(* CODESYS project ctrlxVirtual.export

Project tree, tasks and I/O mapping:
  Device : ctrlX COREvirtual, Bosch Rexroth AG, order no. dependent on customer specific configuration, version 1.14.0.0
    application Application
      libraries: ; SampleSchema, 0.0.1 (Bosch Rexroth)
      task MainTask (cyclic, interval 200 ms, priority 30) calls PLC_PRG
      CheckFunctions/
        function CheckDivDInt [ST]
        function CheckDivLInt [ST]
        function CheckDivLReal [ST]
        function CheckDivReal [ST]
        function CheckLRangeSigned [ST]
        function CheckLRangeUnsigned [ST]
        function CheckRangeSigned [ST]
        function CheckRangeUnsigned [ST]
        function CheckBounds [ST]
        function CheckPointer [ST]
      program PLC_PRG [ST]
    Realtime_Data : DataLayer, Bosch Rexroth AG, version 1.8.0.0
*)

// Device/Application/PLC_PRG
PROGRAM PLC_PRG
VAR
	bStart_read: BOOL := TRUE;
	bStart_write: BOOL;

	// Read values
	bExecute_read: BOOL;
	fbDL_ReadNodeValue: sampleSchema.DL_ReadNodeValue;
	bActive_read: BOOL;
	bDone_read: BOOL;
	
	DataRead: sampleSchema.DL_NodeValue;
	bErrorRead: BOOL;
	ErrorIDRead: ERROR_CODE;
	ErrorIdent_read: ERROR_STRUCT;

	fbR_TRIG_read: R_TRIG;

	fbFlatbuffer : sampleSchema.sample_schema_InertialValue;

	iRead_X: INT;
	iRead_Y: INT;
	iRead_Z: INT;
	iRead: INT;
	
	///Write values
	fbBuilder: sampleSchema.FlatBufferBuilder();
	
	iWrite_X: INT;
	iWrite_Y: INT;
	iWrite_Z: INT;
	iWritten: INT;
	
	bExecute_write: BOOL;
	fbDL_WriteNodeValue: sampleSchema.DL_WriteNodeValue;
	bActive_write: BOOL;
	bDone_write: BOOL;
	fbValueIn: sampleSchema.DL_NodeValue;
	fbValueOut: sampleSchema.DL_NodeValue;
	bError_write: BOOL;
	ErrorID_write: ERROR_CODE;
	ErrorIdent_write: ERROR_STRUCT;
	
	fbR_TRIG_write: R_TRIG;
	

	strNodePath: STRING(255) := 'sdk-cpp-alldata/dynamic/fbs';
	
END_VAR

IF bStart_read THEN
	bStart_read := FALSE;
	bExecute_read := TRUE;	
END_IF


fbDL_ReadNodeValue(
	Execute:= bExecute_read,
	Done=> bDone_read,
	Active=> bActive_read,
	Error=> bErrorRead,
	ErrorID=> ErrorIDRead,
	ErrorIdent=> ErrorIdent_read,
	ClientId:= ,
	NodeName:= strNodePath,
	NodeValue:= DataRead);

IF bDone_read AND bExecute_read THEN
	bExecute_read := FALSE;

	fbFlatbuffer.getRootAsInertialValue(data:=
	DataRead.GetData(), size:= DataRead.GetSize());
	
	iRead_X := fbFlatbuffer.getX();
	iRead_Y := fbFlatbuffer.getY();
	iRead_Z := fbFlatbuffer.getZ();	
	iRead := iRead + 1;
		
	bStart_write := TRUE;
END_IF

	
IF bStart_write THEN
	bStart_write := FALSE;

	iWrite_X := iRead_X + 100;
	iWrite_Y := iRead_Y + 100;
	iWrite_Z := iRead_Z + 100;

	fbBuilder(forceDefaults := TRUE);
	fbFlatbuffer.startInertialValue(fbBuilder);
	fbFlatbuffer.addX(iWrite_X);
	fbFlatbuffer.addY(iWrite_Y);
	fbFlatbuffer.addZ(iWrite_Z);
	fbBuilder.finish(fbFlatbuffer.endInertialValue());
	fbValueIn.SetFlatbuffer(fbBuilder);
	
	bExecute_write := TRUE;
END_IF

	
fbDL_WriteNodeValue(
	Execute:= bExecute_write,
	Done=> bDone_write,
	Active=> bActive_write,
	Error=> bError_write,
	ErrorID=> ErrorID_write,
	ErrorIdent=> ErrorIdent_write,
	ClientId:= ,
	NodeName:= strNodePath,
	NodeValueIn:= fbValueIn,
	NodeValueOut:= fbValueOut);

IF bDone_write AND bExecute_write THEN
	bExecute_write := FALSE;	
	iWritten := iWritten + 1;
	
	bStart_read := TRUE;
END_IF

END_PROGRAM

// Device/Application/CheckFunctions/CheckDivDInt
// Short description:        Test function to increase machine safety by detecting unauthorized division by zero of INT, UINT, DINT, UDINT, WORD and DWORD variables
// 
// Functional description:   This function will be called implicitly before the division takes places.
//                           The divisor will be checked for 0.
//                           In case of 0, an error is entered in the plc logger and the application is stopped due to an access violation to avoid machine damage.
//                           In this case, check the callstack (menu Debug/Callstack) and modify the faulty logic. 
// 
// Handling particularities: This function increases the cycle time of all tasks using divisions.
//                           The increase depends on the number of the divisions.
//                           After inserting/removing this function, no online-change will be possible! 
//                           A complete download will be necessary!
//                           The implementation has to be adjusted to your application/machine.
//                           In case of a division by zero, the PLC-Task will generate an access violation which leads to an application stop.
//                           Please verify whether this default behaviour can damage your machine or lead to a complex recommissioning. 
//                           In this case, adapt the error reaction to your application.
//                          
//                           If your application isn't too time-critical, you should leave this function whil comissioning the machine and production in your application.  
//                           If you remove this function, ensure that your code is faultless.
//                          
// Do not change the declaration of this function! Add only local variables.  
// Do not change the attributes above the function header!
{attribute 'check_div_int32'}
{attribute 'no_check'}
{attribute 'signature_flag' := '1073741824'}
FUNCTION CheckDivDInt : DINT
VAR_INPUT
  divisor: DINT; // Divisor of the division
END_VAR
VAR
  ptNull: POINTER TO BYTE := 0; // Nullpointer for triggering an access violation
  strError: STRING;             // Diagnostic text for the PLC logger entry
END_VAR

    (**************************************************************************************************)
    (* The implementation has to be adjusted to your application/machine.                             *)
    (* This is an exemplary implementation of the function.                                           *)
    (* Per default, an access violation is generated to avoid machine damage                          *)
    (* Check the Call Stack (menu Debug/Callstack) and modify the faulty logic!                       *)
    (**************************************************************************************************)

IF divisor = 0 THEN
  strError:= 'CheckDivDInt: Invalid division by 0 - check the callstack';
//  Default implementation for APPLICATION WILL BE STOPPED: 
//  Set an error into the plc logger
  LogAdd2(hLogger:= CmpLog.LOG_STD_LOGGER,udiCmpID:= 16#1000,udiClassID:= LogClass.LOG_ERROR,udiErrorID:= 1,udiInfoID:= 1,pszInfo:= strError);
//  Triggering an access violation --> Application will be stopped
  ptNull^ := 0;(* Triggering an access violation *)

// // Example for APPLICATION WILL NOT BE STOPPED:
// // Set the divisor to 1 
// //   --> no access violation (div by zero) will be triggered
// //   --> keep PLC-task running 
// // Set a warning into the plc logger
// // NOTE: There is still an implementation error in your application code!
// 
//  LogAdd2(hLogger:= CmpLog.LOG_STD_LOGGER,udiCmpID:= 16#1000,udiClassID:= LogClass.LOG_WARNING,udiErrorID:= 1,udiInfoID:= 1,pszInfo:= strError);
//  CheckDivDint := 1; //Division by 1 instead of zero 
//  return;	

ELSE // division is ok
  CheckDivDInt:=divisor;
END_IF;

END_FUNCTION

// Device/Application/CheckFunctions/CheckDivLInt
// Short description:        Test function to increase machine safety by detecting unauthorized division by zero of LINT, ULINT and LWORD variables
// 
// Functional description:   This function will be called implicitly before the division takes places.
//                           The divisor will be checked for 0.
//                           In case of 0, an error is entered in the plc logger and the application is stopped due to an access violation to avoid machine damage.
//                           In this case, check the callstack (menu Debug/Callstack) and modify the faulty logic. 
// 
// Handling particularities: This function increases the cycle time of all tasks using divisions.
//                           The increase depends on the number of the divisions.
//                           After inserting/removing this function, no online-change will be possible! 
//                           A complete download will be necessary!
//                           The implementation has to be adjusted to your application/machine.
//                           In case of a division by zero, the PLC-Task will generate an access violation which leads to an application stop.
//                           Please verify whether this default behaviour can damage your machine or lead to a complex recommissioning. 
//                           In this case, adapt the error reaction to your application.
//                          
//                           If your application isn't too time-critical, you should leave this function whil comissioning the machine and production in your application.  
//                           If you remove this function, ensure that your code is faultless.
//                          
// Do not change the declaration of this function! Add only local variables.  
// Do not change the attributes above the function header!
{attribute 'check_div_int64'}
{attribute 'no_check'}
{attribute 'signature_flag' := '1073741824'}
FUNCTION CheckDivLInt : LINT
VAR_INPUT
  divisor: LINT; // Divisor of the division
END_VAR
VAR
  ptNull: POINTER TO BYTE := 0; // Nullpointer for triggering an access violation
  strError: STRING;             // Diagnostic text for the PLC logger entry
END_VAR

    (**************************************************************************************************)
    (* The implementation has to be adjusted to your application/machine.                             *)
    (* This is an exemplary implementation of the function.                                           *)
    (* Per default, an access violation is generated to avoid machine damage                          *)
    (* Check the Call Stack (menu Debug/Callstack) and modify the faulty logic!                       *)
    (**************************************************************************************************)

IF divisor = 0 THEN
  strError:= 'CheckDivLInt: Invalid division by 0 - check the callstack';
//  Default implementation for APPLICATION WILL BE STOPPED: 
//  Set an error into the plc logger
  LogAdd2(hLogger:= CmpLog.LOG_STD_LOGGER,udiCmpID:= 16#1000,udiClassID:= LogClass.LOG_ERROR,udiErrorID:= 1,udiInfoID:= 1,pszInfo:= strError);
//  Triggering an access violation --> Application will be stopped
  ptNull^ := 0;(* Triggering an access violation *)

// // Example for APPLICATION WILL NOT BE STOPPED:
// // Set the divisor to 1 
// //   --> no access violation (div by zero) will be triggered
// //   --> keep PLC-task running 
// // Set a warning into the plc logger
// // NOTE: There is still an implementation error in your application code!
//  
//  LogAdd2(hLogger:= CmpLog.LOG_STD_LOGGER,udiCmpID:= 16#1000,udiClassID:= LogClass.LOG_WARNING,udiErrorID:= 1,udiInfoID:= 1,pszInfo:= strError);
//  CheckDivLInt := 1; //Division by 1 instead of zero 
//  return;	

ELSE // division is ok
  CheckDivLInt:=divisor;
END_IF;

END_FUNCTION

// Device/Application/CheckFunctions/CheckDivLReal
// Short description:        Test function to increase machine safety by detecting unauthorized division by zero of variables of type LREAL
// 
// Functional description:   This function will be called implicitly before the division takes places.
//                           The divisor will be checked for 0.0.
//                           In case of 0.0, an error is entered in the plc logger and the application is stopped due to an access violation to avoid machine damage.
//                           In this case, check the callstack (menu Debug/Callstack) and modify the faulty logic. 
// 
// Handling particularities: This function increases the cycle time of all tasks using divisions.
//                           The increase depends on the number of the divisions.
//                           After inserting/removing this function, no online-change will be possible! 
//                           A complete download will be necessary!
//                           The implementation has to be adjusted to your application/machine.
//                           In case of a division by zero, the PLC-Task will generate an access violation which leads to an application stop.
//                           Please verify whether this default behaviour can damage your machine or lead to a complex recommissioning. 
//                           In this case, adapt the error reaction to your application.
//                          
//                           If your application isn't too time-critical, you should leave this function whil comissioning the machine and production in your application.  
//                           If you remove this function, ensure that your code is faultless.
//                          
// Do not change the declaration of this function! Add only local variables.  
// Do not change the attributes above the function header!
{attribute 'check_div_real64'}
{attribute 'no_check'}
{attribute 'signature_flag' := '1073741824'}
FUNCTION CheckDivLReal : LREAL
VAR_INPUT
  divisor: LREAL; // Divisor of the division
END_VAR
VAR
  ptNull: POINTER TO BYTE := 0; // Nullpointer for triggering an access violation
  strError: STRING;             // Diagnostic text for the PLC logger entry
END_VAR

    (**************************************************************************************************)
    (* The implementation has to be adjusted to your application/machine.                             *)
    (* This is an exemplary implementation of the function.                                           *)
    (* Per default, an access violation is generated to avoid machine damage                          *)
    (* Check the Call Stack (menu Debug/Callstack) and modify the faulty logic!                       *)
    (**************************************************************************************************)

IF divisor = 0 THEN
  strError:= 'CheckDivLReal: Invalid division by 0 - check the callstack';
//  Default implementation for APPLICATION WILL BE STOPPED: 
//  Set an error into the plc logger
  LogAdd2(hLogger:= CmpLog.LOG_STD_LOGGER,udiCmpID:= 16#1000,udiClassID:= LogClass.LOG_ERROR,udiErrorID:= 1,udiInfoID:= 1,pszInfo:= strError);
//  Triggering an access violation --> Application will be stopped
  ptNull^ := 0;(* Triggering an access violation *)

// // Example for APPLICATION WILL NOT BE STOPPED:
// // Set the divisor to 1.0 
// //   --> no access violation (div by zero) will be triggered
// //   --> keep PLC-task running 
// // Set a warning into the plc logger
// // NOTE: There is still an implementation error in your application code!
//
//  LogAdd2(hLogger:= CmpLog.LOG_STD_LOGGER,udiCmpID:= 16#1000,udiClassID:= LogClass.LOG_WARNING,udiErrorID:= 1,udiInfoID:= 1,pszInfo:= strError);
//  CheckDivLReal := 1.0; //Division by 1 instead of zero 
//  return;	

ELSE // division is ok
  CheckDivLReal:=divisor;
END_IF;

END_FUNCTION

// Device/Application/CheckFunctions/CheckDivReal
// Short description:        Test function to increase machine safety by detecting unauthorized division by zero of variables of type REAL. 
// 
// Functional description:   This function will be called implicitly before the division takes places.
//                           The divisor will be checked for 0.0.
//                           In case of 0.0, an error is entered in the plc logger and the application is stopped due to an access violation to avoid machine damage.
//                           In this case, check the callstack (menu Debug/Callstack) and modify the faulty logic. 
// 
// Handling particularities: This function increases the cycle time of all tasks using divisions.
//                           The increase depends on the number of the divisions.
//                           After inserting/removing this function, no online-change will be possible! 
//                           A complete download will be necessary!
//                           The implementation has to be adjusted to your application/machine.
//                           In case of a division by zero, the PLC-Task will generate an access violation which leads to an application stop.
//                           Please verify whether this default behaviour can damage your machine or lead to a complex recommissioning. 
//                           In this case, adapt the error reaction to your application.
//                          
//                           If your application isn't too time-critical, you should leave this function whil comissioning the machine and production in your application.  
//                           If you remove this function, ensure that your code is faultless.
//                          
// Do not change the declaration of this function! Add only local variables.  
// Do not change the attributes above the function header!
{attribute 'check_div_real32'}
{attribute 'no_check'}
{attribute 'signature_flag' := '1073741824'}
FUNCTION CheckDivReal : REAL
VAR_INPUT
  divisor: REAL; // Divisor of the division
END_VAR
VAR
  ptNull: POINTER TO BYTE := 0; // Nullpointer for triggering an access violation
  strError: STRING;             // Diagnostic text for the PLC logger entry
END_VAR

    (**************************************************************************************************)
    (* The implementation has to be adjusted to your application/machine.                             *)
    (* This is an exemplary implementation of the function.                                           *)
    (* Per default, an access violation is generated to avoid machine damage                          *)
    (* Check the Call Stack (menu Debug/Callstack) and modify the faulty logic!                       *)
    (**************************************************************************************************)

IF divisor = 0 THEN
  strError:= 'CheckDivReal: Invalid division by 0 - check the callstack';
//  Default implementation for APPLICATION WILL BE STOPPED: 
//  Set an error into the plc logger
  LogAdd2(hLogger:= CmpLog.LOG_STD_LOGGER,udiCmpID:= 16#1000,udiClassID:= LogClass.LOG_ERROR,udiErrorID:= 1,udiInfoID:= 1,pszInfo:= strError);
//  Triggering an access violation --> Application will be stopped
  ptNull^ := 0;(* Triggering an access violation *)

// // Example for APPLICATION WILL NOT BE STOPPED:
// // Set the divisor to 1 
// //   --> no access violation (div by zero) will be triggered
// //   --> keep PLC-task running 
// // Set a warning into the plc logger
// // NOTE: There is still an implementation error in your application code!
// 
//  LogAdd2(hLogger:= CmpLog.LOG_STD_LOGGER,udiCmpID:= 16#1000,udiClassID:= LogClass.LOG_WARNING,udiErrorID:= 1,udiInfoID:= 1,pszInfo:= strError);
//  CheckDivReal := 1.0; //Division by 1 instead of zero 
//  return;	

ELSE // division is ok
  CheckDivReal:=divisor;
END_IF;

END_FUNCTION

// Device/Application/CheckFunctions/CheckLRangeSigned
// Short description:        Test function to increase machine safety by checking if value is within signed range (LINT) 
// 
// Functional description:  This function will be called implicitly before any access to range signed values.
//                           In case of invalid access, an error is entered in the diagnostic logbook and the application is stopped due to an access violation to avoid machine damage.
//                           In this case, check the callstack (menu Debug/Callstack) and modify the faulty logic. 
//                          
// Handling particularities: This function increases the cycle time of all tasks accessing range signed values. 
//                           The increase depends on the number of the read/write accesses.
// 
//                           After inserting/removing this function, no online-change will be possible! 
//                           A complete download will be necessary!
//                           The implementation has to be adjusted to your application/machine.
//                           In case of a division by zero, the PLC-Task will generate an access violation which leads to an application stop.
//                           Please verify whether this default behaviour can damage your machine or lead to a complex recommissioning. 
//                           In this case, adapt the error reaction to your application.
//
//                           If your application isn't too time-critical, you should leave this function whil comissioning the machine and production in your application.  
//                           If you remove this function, ensure that your code is faultless.
//                          
// Do not change the declaration of this function! Add only local variables.  
// Do not change the attributes above the function header!
{attribute 'no_check'}
{attribute 'check_lrange_signed'}
{attribute 'signature_flag' := '1073741824'}
FUNCTION CheckLRangeSigned : LINT
VAR_INPUT
  value: LINT;
  lower: LINT;
  upper: LINT;
END_VAR
VAR
  ptNull: POINTER TO BYTE := 0; // Nullpointer for triggering an access violation
  strError: STRING;             // Diagnostic text for the PLC logger entry
END_VAR

    (**************************************************************************************************)
    (* The implementation has to be adjusted to your application/machine.                             *)
    (* This is an exemplary implementation of the function.                                           *)
    (* Per default, an access violation is generated to avoid machine damage                          *)
    (* Check the Call Stack (menu Debug/Callstack) and modify the faulty logic!                       *)
    (**************************************************************************************************)

IF (value < lower) THEN
  strError:= 'CheckLRangeSigned: Lower value ';
  strError:=CONCAT(STR1:=strError  , STR2:= LINT_TO_STRING(lower));
  strError:=CONCAT(STR1:=strError  , STR2:= ' underrunned by ');
  strError:=CONCAT(STR1:=strError  , STR2:= LINT_TO_STRING(value));
//  Default implementation for APPLICATION WILL BE STOPPED: 
//  Set an error into the plc logger
  LogAdd2(hLogger:= CmpLog.LOG_STD_LOGGER,udiCmpID:= 16#1000,udiClassID:= LogClass.LOG_ERROR,udiErrorID:= 1,udiInfoID:= 1,pszInfo:= strError);
//  Triggering an access violation --> Application will be stopped
  ptNull^ := 0;(* Triggering an access violation *)

// // Example for APPLICATION WILL NOT BE STOPPED:
// // Limit the faulty value to the lower value 
// // Set a warning into the plc logger
// // NOTE: There is still an implementation error in your application code!
//
//	LogAdd2(hLogger:= CmpLog.LOG_STD_LOGGER,udiCmpID:= 16#1000,udiClassID:= LogClass.LOG_WARNING,udiErrorID:= 1,udiInfoID:= 1,pszInfo:= strError);
// 	CheckLRangeSigned := lower; //set value to lower value
//  return;
  
ELSIF(value > upper) THEN
  strError:= 'CheckLRangeSigned: Upper value ';
  strError:=CONCAT(STR1:=strError  , STR2:= LINT_TO_STRING(upper));
  strError:=CONCAT(STR1:=strError  , STR2:= ' overrunned by ');
  strError:=CONCAT(STR1:=strError  , STR2:= LINT_TO_STRING(value));

//  Default implementation for APPLICATION WILL BE STOPPED: 
//  Set an error into the plc logger
  LogAdd2(hLogger:= CmpLog.LOG_STD_LOGGER,udiCmpID:= 16#1000,udiClassID:= LogClass.LOG_ERROR,udiErrorID:= 1,udiInfoID:= 1,pszInfo:= strError);
//  Triggering an access violation --> Application will be stopped
  ptNull^ := 0;(* Triggering an access violation *)

// // Example for APPLICATION WILL NOT BE STOPPED:
// // Limit the faulty value to the upper value 
// // Set a warning into the plc logger
// // NOTE: There is still an implementation error in your application code!
// 
//  LogAdd2(hLogger:= CmpLog.LOG_STD_LOGGER,udiCmpID:= 16#1000,udiClassID:= LogClass.LOG_WARNING,udiErrorID:= 1,udiInfoID:= 1,pszInfo:= strError);
//  CheckLRangeSigned := upper; //set value to upper value
//  return;	

ELSE // value ist within valid range
  CheckLRangeSigned := value;
END_IF

END_FUNCTION

// Device/Application/CheckFunctions/CheckLRangeUnsigned
// Short description:        Test function to increase machine safety by checking if value is within unsigned range  (ULINT, LWORD) 
// 
// Functional description:   This function will be called implicitly before any access to range signed values.
//                           In case of invalid access, an error is entered in the diagnostic logbook and the application is stopped due to an access violation to avoid machine damage.
//                           In this case, check the callstack (menu Debug/Callstack) and modify the faulty logic. 
//                          
// Handling particularities: This function increases the cycle time of all tasks accessing range signed values. 
//                           The increase depends on the number of the read/write accesses.
// 
//                           After inserting/removing this function, no online-change will be possible! 
//                           A complete download will be necessary!
//                           The implementation has to be adjusted to your application/machine.
//                           In case of a division by zero, the PLC-Task will generate an access violation which leads to an application stop.
//                           Please verify whether this default behaviour can damage your machine or lead to a complex recommissioning. 
//                           In this case, adapt the error reaction to your application.
//                          
//                           If your application isn't too time-critical, you should leave this function whil comissioning the machine and production in your application.  
//                           If you remove this function, ensure that your code is faultless.
//                          
// Do not change the declaration of this function! Add only local variables.  
// Do not change the attributes above the function header!
{attribute 'no_check'}
{attribute 'check_lrange_unsigned'}
{attribute 'signature_flag' := '1073741824'}
FUNCTION CheckLRangeUnsigned : ULINT
VAR_INPUT
  value: ULINT;
  lower: ULINT;
  upper: ULINT;
END_VAR
VAR
  ptNull: POINTER TO BYTE := 0; // Nullpointer for triggering an access violation
  strError: STRING;             // Diagnostic text for the PLC logger entry
END_VAR

    (**************************************************************************************************)
    (* The implementation has to be adjusted to your application/machine.                             *)
    (* This is an exemplary implementation of the function.                                           *)
    (* Per default, an access violation is generated to avoid machine damage                          *)
    (* Check the Call Stack (menu Debug/Callstack) and modify the faulty logic!                       *)
    (**************************************************************************************************)

IF (value < lower) THEN
  strError:= 'CheckLRangeUnsigned: Lower value ';
  strError:=CONCAT(STR1:=strError  , STR2:= ULINT_TO_STRING(lower));
  strError:=CONCAT(STR1:=strError  , STR2:= ' underrunned by ');
  strError:=CONCAT(STR1:=strError  , STR2:= ULINT_TO_STRING(value));
//  Default implementation for APPLICATION WILL BE STOPPED: 
//  Set an error into the plc logger
  LogAdd2(hLogger:= CmpLog.LOG_STD_LOGGER,udiCmpID:= 16#1000,udiClassID:= LogClass.LOG_ERROR,udiErrorID:= 1,udiInfoID:= 1,pszInfo:= strError);
//  Triggering an access violation --> Application will be stopped
  ptNull^ := 0;(* Triggering an access violation *)

// // Example for APPLICATION WILL NOT BE STOPPED:
// // Limit the faulty value to the lower value 
// // Set a warning into the plc logger
// // NOTE: There is still an implementation error in your application code!
// 
//  CheckLRangeUnsigned := lower; //set value to lower value
//  return;

ELSIF(value > upper) THEN
  strError:= 'CheckLRangeUnsigned: Upper value ';
  strError:=CONCAT(STR1:=strError  , STR2:= ULINT_TO_STRING(upper));
  strError:=CONCAT(STR1:=strError  , STR2:= ' overrunned by ');
  strError:=CONCAT(STR1:=strError  , STR2:= ULINT_TO_STRING(value));

//  Default implementation for APPLICATION WILL BE STOPPED: 
//  Set an error into the plc logger
 LogAdd2(hLogger:= CmpLog.LOG_STD_LOGGER,udiCmpID:= 16#1000,udiClassID:= LogClass.LOG_ERROR,udiErrorID:= 1,udiInfoID:= 1,pszInfo:= strError);
//  Triggering an access violation --> Application will be stopped
 ptNull^ := 0;(* Triggering an access violation *)

// // Example for APPLICATION WILL NOT BE STOPPED:
// // Limit the faulty value to the upper value 
// // Set a warning into the plc logger
// // NOTE: There is still an implementation error in your application code!
// 
//  LogAdd2(hLogger:= CmpLog.LOG_STD_LOGGER,udiCmpID:= 16#1000,udiClassID:= LogClass.LOG_WARNING,udiErrorID:= 1,udiInfoID:= 1,pszInfo:= strError);
//  CheckLRangeUnsigned := upper; //set value to upper value
//  return;	

ELSE // value ist within valid range
  CheckLRangeUnsigned := value;
END_IF

END_FUNCTION

// Device/Application/CheckFunctions/CheckRangeSigned
// Short description:        Test function to increase machine safety by checking if value is within signed range (INT, DINT)  
// 
// Functional description:   This function will be called implicitly before any access to range signed values.
//                           In case of invalid access, an error is entered in the diagnostic logbook and the application is stopped due to an access violation to avoid machine damage.
//                           In this case, check the callstack (menu Debug/Callstack) and modify the faulty logic. 
//                          
// Handling particularities: This function increases the cycle time of all tasks accessing range signed values. 
//                           The increase depends on the number of the read/write accesses.
// 
//                           After inserting/removing this function, no online-change will be possible! 
//                           A complete download will be necessary!
//                           The implementation has to be adjusted to your application/machine.
//                           In case of a division by zero, the PLC-Task will generate an access violation which leads to an application stop.
//                           Please verify whether this default behaviour can damage your machine or lead to a complex recommissioning. 
//                           In this case, adapt the error reaction to your application.
//                          
//                           If your application isn't too time-critical, you should leave this function whil comissioning the machine and production in your application.  
//                           If you remove this function, ensure that your code is faultless.
//                          
// Do not change the declaration of this function! Add only local variables.  
// Do not change the attributes above the function header!
{attribute 'no_check'}
{attribute 'check_range_signed'}
{attribute 'signature_flag' := '1073741824'}
FUNCTION CheckRangeSigned : DINT
VAR_INPUT
  value: DINT;
  lower: DINT;
  upper: DINT;
END_VAR
VAR
  ptNull: POINTER TO BYTE := 0; // Nullpointer for triggering an access violation
  strError: STRING;             // Diagnostic text for the PLC logger entry
END_VAR

    (**************************************************************************************************)
    (* The implementation has to be adjusted to your application/machine.                             *)
    (* This is an exemplary implementation of the function.                                           *)
    (* Per default, an access violation is generated to avoid machine damage                          *)
    (* Check the Call Stack (menu Debug/Callstack) and modify the faulty logic!                       *)
    (**************************************************************************************************)

IF (value < lower) THEN
  strError:= 'CheckRangeSigned: Lower value ';
  strError:=CONCAT(STR1:=strError  , STR2:= DINT_TO_STRING(lower));
  strError:=CONCAT(STR1:=strError  , STR2:= ' underrunned by ');
  strError:=CONCAT(STR1:=strError  , STR2:= DINT_TO_STRING(value));
//  Default implementation for APPLICATION WILL BE STOPPED: 
//  Set an error into the plc logger
  LogAdd2(hLogger:= CmpLog.LOG_STD_LOGGER,udiCmpID:= 16#1000,udiClassID:= LogClass.LOG_ERROR,udiErrorID:= 1,udiInfoID:= 1,pszInfo:= strError);
//  Triggering an access violation --> Application will be stopped
  ptNull^ := 0;(* Triggering an access violation *)

// // Example for APPLICATION WILL NOT BE STOPPED:
// // Limit the faulty value to the lower value 
// // Set a warning into the plc logger
// // NOTE: There is still an implementation error in your application code!
//
//  LogAdd2(hLogger:= CmpLog.LOG_STD_LOGGER,udiCmpID:= 16#1000,udiClassID:= LogClass.LOG_WARNING,udiErrorID:= 1,udiInfoID:= 1,pszInfo:= strError);
//  CheckRangeSigned := lower; //set value to lower value
//  return;

ELSIF(value > upper) THEN
  strError:= 'CheckRangeSigned: Upper value ';
  strError:=CONCAT(STR1:=strError  , STR2:= DINT_TO_STRING(upper));
  strError:=CONCAT(STR1:=strError  , STR2:= ' overrunned by ');
  strError:=CONCAT(STR1:=strError  , STR2:= DINT_TO_STRING(value));

//  Default implementation for APPLICATION WILL BE STOPPED: 
//  Set an error into the plc logger
  LogAdd2(hLogger:= CmpLog.LOG_STD_LOGGER,udiCmpID:= 16#1000,udiClassID:= LogClass.LOG_ERROR,udiErrorID:= 1,udiInfoID:= 1,pszInfo:= strError);
//  Triggering an access violation --> Application will be stopped
  ptNull^ := 0;(* Triggering an access violation *)

// // Example for APPLICATION WILL NOT BE STOPPED:
// // Limit the faulty value to the upper value 
// // Set a warning into the plc logger
// // NOTE: There is still an implementation error in your application code!
// 
//  LogAdd2(hLogger:= CmpLog.LOG_STD_LOGGER,udiCmpID:= 16#1000,udiClassID:= LogClass.LOG_WARNING,udiErrorID:= 1,udiInfoID:= 1,pszInfo:= strError);
//  CheckRangeSigned := upper; //set value to upper value
//  return;	

ELSE // value ist within valid range
  CheckRangeSigned := value;
END_IF

END_FUNCTION

// Device/Application/CheckFunctions/CheckRangeUnsigned
// Short description:        Test function to increase machine safety by checking if value is within unsigned range (UINT, UDINT, WORD, DWORD)
// 
// Functional description:   This function will be called implicitly before any access to range unsigned values.
//                           In case of invalid access, an error is entered in the diagnostic logbook and the application is stopped due to an access violation to avoid machine damage.
//                           In this case, check the callstack (menu Debug/Callstack) and modify the faulty logic. 
//                          
// Handling particularities: This function increases the cycle time of all tasks accessing range signed values. 
//                           The increase depends on the number of the read/write accesses.
// 
//                           After inserting/removing this function, no online-change will be possible! 
//                           A complete download will be necessary!
//                           The implementation has to be adjusted to your application/machine.
//                           In case of a division by zero, the PLC-Task will generate an access violation which leads to an application stop.
//                           Please verify whether this default behaviour can damage your machine or lead to a complex recommissioning. 
//                           In this case, adapt the error reaction to your application.
//                          
//                           If your application isn't too time-critical, you should leave this function whil comissioning the machine and production in your application.  
//                           If you remove this function, ensure that your code is faultless.
//                          
// Do not change the declaration of this function! Add only local variables.  
// Do not change the attributes above the function header!
{attribute 'check_range_unsigned'}
{attribute 'signature_flag' := '1073741824'}
{attribute 'no_check'}
FUNCTION CheckRangeUnsigned : UDINT
VAR_INPUT
  value: UDINT;
  lower: UDINT;
  upper: UDINT;
END_VAR
VAR
  ptNull: POINTER TO BYTE := 0; // Nullpointer for triggering an access violation
  strError: STRING;             // Diagnostic text for the PLC logger entry
END_VAR

    (**************************************************************************************************)
    (* The implementation has to be adjusted to your application/machine.                             *)
    (* This is an exemplary implementation of the function.                                           *)
    (* Per default, an access violation is generated to avoid machine damage                          *)
    (* Check the Call Stack (menu Debug/Callstack) and modify the faulty logic!                       *)
    (**************************************************************************************************)

IF (value < lower) THEN
  strError:= 'CheckRangeUnsigned: Lower value ';
  strError:=CONCAT(STR1:=strError  , STR2:= UDINT_TO_STRING(lower));
  strError:=CONCAT(STR1:=strError  , STR2:= ' underrunned by ');
  strError:=CONCAT(STR1:=strError  , STR2:= UDINT_TO_STRING(value));
//  Default implementation for APPLICATION WILL BE STOPPED: 
//  Set an error into the plc logger
  LogAdd2(hLogger:= CmpLog.LOG_STD_LOGGER,udiCmpID:= 16#1000,udiClassID:= LogClass.LOG_ERROR,udiErrorID:= 1,udiInfoID:= 1,pszInfo:= strError);
//  Triggering an access violation --> Application will be stopped
  ptNull^ := 0;(* Triggering an access violation *)

// // Example for APPLICATION WILL NOT BE STOPPED:
// // Limit the faulty value to the lower value 
// // Set a warning into the plc logger
// // NOTE: There is still an implementation error in your application code!
//
//  LogAdd2(hLogger:= CmpLog.LOG_STD_LOGGER,udiCmpID:= 16#1000,udiClassID:= LogClass.LOG_WARNING,udiErrorID:= 1,udiInfoID:= 1,pszInfo:= strError);
//  CheckRangeUnsigned := lower; //set value to lower value
//  return;

ELSIF(value > upper) THEN
  strError:= 'CheckRangeUnsigned: Upper value ';
  strError:=CONCAT(STR1:=strError  , STR2:= UDINT_TO_STRING(upper));
  strError:=CONCAT(STR1:=strError  , STR2:= ' overrunned by ');
  strError:=CONCAT(STR1:=strError  , STR2:= UDINT_TO_STRING(value));

//  Default implementation for APPLICATION WILL BE STOPPED: 
//  Set an error into the plc logger
  LogAdd2(hLogger:= CmpLog.LOG_STD_LOGGER,udiCmpID:= 16#1000,udiClassID:= LogClass.LOG_ERROR,udiErrorID:= 1,udiInfoID:= 1,pszInfo:= strError);
//  Triggering an access violation --> Application will be stopped
 ptNull^ := 0;(* Triggering an access violation *)

// // Example for APPLICATION WILL NOT BE STOPPED:
// // Limit the faulty value to the upper value 
// // Set a warning into the plc logger
// // NOTE: There is still an implementation error in your application code!
// 
//  LogAdd2(hLogger:= CmpLog.LOG_STD_LOGGER,udiCmpID:= 16#1000,udiClassID:= LogClass.LOG_WARNING,udiErrorID:= 1,udiInfoID:= 1,pszInfo:= strError);
//  CheckRangeUnsigned := upper; //set value to upper value
//  return;

ELSE // value ist within valid range
  CheckRangeUnsigned := value;
END_IF

END_FUNCTION

// Device/Application/CheckFunctions/CheckBounds
// Short description:      Test function to increase machine safety by checking for unauthorized array indices accesses.
// 
// Functional description: This function is implicitly called prior to each array access and verifies if the access is within the valid array bounds.
//                         If the access is authorized, the function returns the index to the calling POU and the access is completed.
//                         If the access is unauthorized, an exception is triggered as default error reaction. This exception results in an application stop and the system is set to safe state. 
//   
// Handling particularities: Sporadically, the implemented default error reaction has TO be adjusted TO the application. 
//                           For example, stopping of the application can be invalid and can result in complicated recommissioning or even injury to people or damage to machines.
//                           Thus, adjust the default error reaction to your application.
//                           After inserting/removing this function in/from the project, no online change is possible.
//                           A complete download is required.
// 
// Further information:    The implicit calls of this check function are realized in all POUs but not in POUs of protected (*.compiled library) 
//                         and open (*.library) libraries or in POUs with the attribute {attribute 'no_check'}. Consequently, they do not increase the runtime.
//                         If the check is also to be performed in open libraries, enter the compiler definition 
//                         checks_in_libs in the field Compiler-Defines of the Build tab in the property dialog of the application node.
//                         An increased runtime depends on the number of programmed array accesses.
// 
//                         To reduce task runtimes, add the attribute 'no_check' to the POUs. 
//                         Checks performed by the check functions (CheckPointer, CheckBounds, CheckDiv, CheckRange) are not performed in these POUs. 
//                         Thus, these POUs have to be checked by the user regarding pointer programming, divisions and array accesses.  
//                         For more information, refer to the F1-help.
// 
//                         In the standard implementation, it is checked if the array access takes place within the valid array boundaries.
// 
//                         In case of invalid access (outside the valid array boundaries), an error is entered in the PLC logger and the application is stopped to avoid injury to persons and damage to machines.
//                         In this case, check the callstack (menu Debug/Callstack) and change the incorrect logic.
//
//                         If your application is not time-critical, use this function during commissioning as well as during the production phase of the machine.
//                         Only remove this function if you are sure that your user code is free from errors!
// 
// Do not change the declaration of this function! Add only local variables.  
// Do not change the attributes above the function header!
{attribute 'check_bounds'}
{attribute 'no_check'}
{attribute 'signature_flag' := '1073741824'}
FUNCTION CheckBounds : DINT
VAR_INPUT
  index, lower, upper: DINT;   // Index of the array, lower bound and upper bound
END_VAR
VAR
  ptNull: POINTER TO BYTE :=0; // Nullpointer for triggering an access violation
  strError: STRING;            // Diagnostic text for the PLC logger entry
END_VAR

    (*****************************************************************************************************)
    (* The implementation has to be adjusted to your application/machine.                                *)
    (* This is an exemplary implementation of the function.                                              *)
    (* Per default, an access violation is generated in case of an faulty acces to avoid machine damage. *)
    (* In this case, check the Call Stack (menu Debug/Callstack) and modify the faulty logic.            *)
    (*****************************************************************************************************)

IF  index < lower THEN 
  strError:= 'CheckBounds: Lower arrayindex ';
  strError:=CONCAT(STR1:=strError  , STR2:= DINT_TO_STRING(lower));
  strError:=CONCAT(STR1:=strError  , STR2:= ' underrunned by ');
  strError:=CONCAT(STR1:=strError  , STR2:= DINT_TO_STRING(index));
//  Default implementation for APPLICATION WILL BE STOPPED: 
//  Set an error into the plc logger
  LogAdd2(hLogger:= CmpLog.LOG_STD_LOGGER,udiCmpID:= 16#1000,udiClassID:= LogClass.LOG_ERROR,udiErrorID:= 1,udiInfoID:= 1,pszInfo:= strError);
//  Triggering an access violation --> Application will be stopped
  ptNull^ := 0;(* Triggering an access violation *)

// // Example for APPLICATION WILL NOT BE STOPPED:
// // Limit the faulty index to the lower index 
// //     --> no memory will be overwritten
// //     --> Keep PLC-task running
// // Set a warning into the plc logger
// // NOTE: There is still an implementation error in your application code!
// //  LogAdd2(hLogger:= CmpLog.LOG_STD_LOGGER,udiCmpID:= 16#1000,udiClassID:= LogClass.LOG_WARNING,udiErrorID:= 1,udiInfoID:= 1,pszInfo:= strError);
// // 
//  CheckBounds := lower; //access to the lower index only 
//  return;

ELSIF  index > upper THEN
  strError:= 'CheckBounds: Higher arrayindex ';
  strError:=CONCAT(STR1:=strError  , STR2:= DINT_TO_STRING(upper));
  strError:=CONCAT(STR1:=strError  , STR2:= ' overrunned by ');
  strError:=CONCAT(STR1:=strError  , STR2:= DINT_TO_STRING(index));

//  Default implementation for APPLICATION WILL BE STOPPED: 
//  Set an error into the plc logger
  LogAdd2(hLogger:= CmpLog.LOG_STD_LOGGER,udiCmpID:= 16#1000,udiClassID:= LogClass.LOG_ERROR,udiErrorID:= 1,udiInfoID:= 1,pszInfo:= strError);
//  Triggering an access violation --> Application will be stopped
  ptNull^ := 0;(* Triggering an access violation *)

// // Example for APPLICATION WILL NOT BE STOPPED:
// // Limit the faulty index to the upper index 
// //     --> no memory will be overwritten
// //     --> Keep PLC-task running
// // Set a warning into the plc logger
// // NOTE: There is still an implementation error in your application code!
//  LogAdd2(hLogger:= CmpLog.LOG_STD_LOGGER,udiCmpID:= 16#1000,udiClassID:= LogClass.LOG_WARNING,udiErrorID:= 1,udiInfoID:= 1,pszInfo:= strError);
// 
//  CheckBounds := upper; //access to the upper index only 
//  return;

ELSE // access to array is within lower and upper index --> ok  
  CheckBounds := index;
END_IF

END_FUNCTION

// Device/Application/CheckFunctions/CheckPointer
// Short description:      Test function to increase machine safety by detecting unauthorized accesses via POINTER and REFERENCE variables
//
// Functional description: This function is implicitly called prior to each pointer access and verifies if the access is invalid to 0.
//                         If the access is authorized, the function returns the pointer to the calling POU and the access is completed.
//                         If the access is unauthorized, an exception is triggered as default error reaction. This exception results in an application stop and the system is set to safe state. 
//                         It is recommended to adapt an appropriate error response to the machine application.
//   
// Handling particularities: Sporadically, the implemented default error reaction has to be adjusted to the application. 
//                           For example, stopping of the application can be invalid and can result in complicated recommissioning or even injury to people or damage to machines.
//                           Thus, adjust the default error reaction to your application.
//                           After inserting/removing this function in/from the project, no online change is possible.
//                           A complete download is required.
//                         
// Further information:    The implicit calls of this check function are realized in all POUs but not in POUs of protected (*.compiled library) 
//                         and open (*.library) libraries or in POUs with the attribute {attribute 'no_check'}. Consequently, they do not increase the runtime.
//                         If the check is also to be performed in open libraries, enter the compiler definition 
//                         checks_in_libs in the field Compiler-Defines of the Build tab in the property dialog of the application node.
//                         An increased runtime depends on the number of programmed pointer accesses or the use of REFERENCE variables.
//                         
//                         To reduce task runtimes, add the attribute 'no_check' to the POUs. 
//                         Checks performed by the check functions (CheckPointer, CheckBounds, CheckDiv, CheckRange) are not performed in these POUs. 
//                         Thus, these POUs have to be checked by the user regarding pointer programming, divisions and array accesses.  
//                         For more information, refer to the F1-help.
//                         
//                         In the standard implementation, it is checked if the pointer access takes place to Adress 16#0 (NULL-Pointer).
//                         In this case, check the callstack (menu Debug/Callstack) and change the incorrect logic.
//                         
//                         If your application is not time-critical, use this function during commissioning as well as during the production phase of the machine.
//                         Only remove this function if you are sure that your user code is free from errors!
//
// Do not change the declaration of this function! Add only local variables.  
// Do not change the attributes above the function header!
{attribute 'check_pointer'}
{attribute 'signature_flag' := '1073741824'}
{attribute 'no_check'}
FUNCTION CheckPointer : POINTER TO BYTE
VAR_INPUT 
  ptToTest : POINTER TO BYTE; // Pointer target address
  iSize : DINT;		            // Size of the type to which the pointer points. (z.B.: 20 für POINTER TO ARRAY [1..10] OF WORD) 
  iGran : DINT;		            // Granularity of the pointer access. This is the size of the largest unstructured data type in the type to which the pointer points. 
                                // (e.g.: 2 for POINTER TO ARRAY [0..9] OF INT).
  bWrite: BOOL;		            // Indicates read or write access. TRUE = write access.
END_VAR
VAR
  ptNull:   POINTER TO BYTE := 0; // Nullpointer for triggering an access violation
  strError: STRING(128);          // Diagnostic text for the PLC logger entry
  i: INT;						              // Index variable
END_VAR

IF ptToTest = 0 THEN //Just check NULL-Pointer

  IF bWrite THEN // write access
    strError:='CheckPointer: Invalid write-access to 16#0';
  ELSE
    strError:='CheckPointer: Invalid read-access to 16#0';
  END_IF
  strError:=CONCAT(STR1:=strError  , STR2:= ' - Size: ');
  strError:=CONCAT(STR1:=strError  , STR2:=TO_STRING(iSize));
  strError:=CONCAT(STR1:=strError  , STR2:=' - See callstack for reason!');
  
  LogAdd2(hLogger:= CmpLog.LOG_STD_LOGGER,udiCmpID:= 16#1000,udiClassID:= LogClass.LOG_ERROR,udiErrorID:= 1,udiInfoID:= 1,pszInfo:= strError);
  //  Triggering an access violation --> Application will be stopped
  //  Sporadically, this default error reaction has to be adjusted to the application. 
  //  For example, stopping of the application can be invalid and can result in complicated recommissioning or even injury to people or damage to machines.
  //  Thus, adjust the default error reaction to your application.
  ptNull^ := 0; //Triggering an access violation 
	
ELSE // pointer is not a NULL-Pointer
	CheckPointer := ptToTest; 
END_IF

END_FUNCTION
